INTERFACE I_AliasDatatypeAddedEvent EXTENDS I_Event

PROPERTY PUBLIC Target : I_AliasDatatype
GET
END_GET
END_PROPERTY

END_INTERFACE

(* stored: Version 1.1.0.1, ProductVersion 3.1.4024.12
   Itf I_AliasDatatypeAddedEvent: Id {c986e168-e397-0724-228c-66b19ba9da4c}
   Property Target: Id {a888a560-c48d-0725-0dfc-138d164bb893}
   Get Get: Id {5e253326-c2e1-0077-3309-a7e95ee90a78} *)
